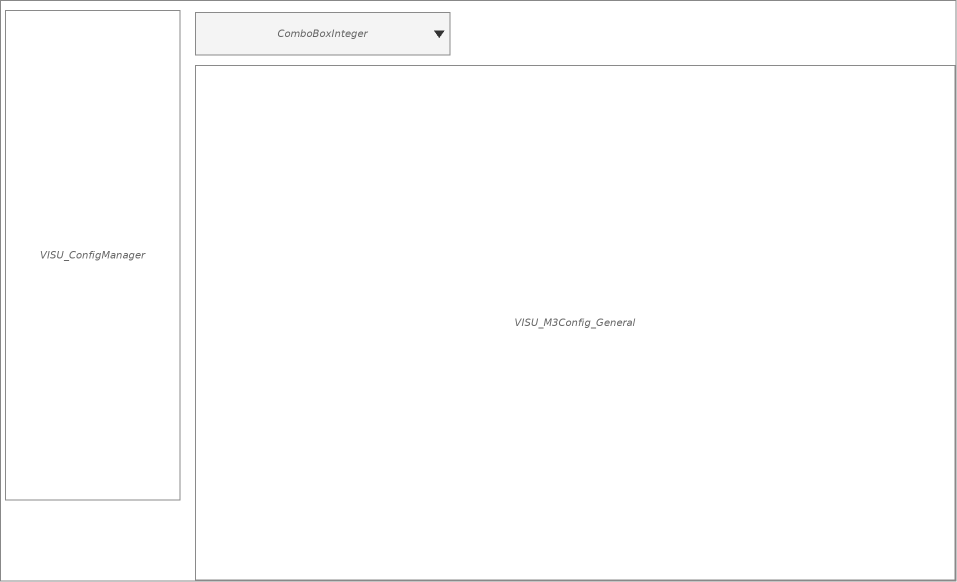
VISUALIZATION VISU_M3Config  // 957x582
VAR_IN_OUT
    m3Widget : M3Widget;
    editableConfig : M3Config;
	activeConfig : M3Config;
    mgr : ConfigManager;
    mgrWidget : ConfigManagerWidget;
END_VAR
    Frame (195,65 760x515), frame switch variable: m3Widget.currentConfigTab
        shows VISU_M3Config_General(active := activeConfig, editable := editableConfig)
        shows VISU_M3Config_KnownPositions(currentPosition := m3Widget.currentConfigTabPosition, active := activeConfig.knownPositions, editable := editableConfig.knownPositions)
        shows VISU_M3Config_Rotation_General(active := activeConfig.rotation, editable := editableConfig.rotation)
        shows VISU_FaulhaberDriveConfig(active := activeConfig.rotation.antiBacklashDrive, editable := editableConfig.rotation.antiBacklashDrive)
        shows VISU_FaulhaberDriveConfig(active := activeConfig.rotation.antiBacklashDrive, editable := editableConfig.rotation.antiBacklashDrive)
        shows VISU_M3Config_Translation_General(active := activeConfig.translation, editable := editableConfig.translation)
        shows VISU_FaulhaberDriveConfig(active := activeConfig.translation.motorDrive, editable := editableConfig.translation.motorDrive)
        p1979262768: mgr
        p1553603785: mgrWidget
    Frame (5,10 175x490)
        shows VISU_ConfigManager(mgr := mgr, widget := mgrWidget)
    ComboBoxInteger (195,12 255x43), variable: m3Widget.currentConfigTab, text list: 'M3ConfigTabsTextList'
END_VISUALIZATION

(* stored: Version 1.1.0.1, ProductVersion 3.1.4019.2
   Visu VISU_M3Config: Id {5d4b07a9-012d-4493-810f-d1458d58db55} *)
